PROGRAM P_EnOcean
VAR
	fbKL6581			: FB_KL6581;
	stKL6581_in  AT %I* : KL6581_INPUT;
	stKL6581_out AT %Q*	: KL6581_OUTPUT;
	stKL6581			: STR_KL6581;
	bInitCom			: BOOL := TRUE;
	
	arrEnOcean_Search	: ARRAY [1..8] OF FB_EnOcean_Search;
	nSearchIdx			: BYTE;
	bSerach				: BOOL;
	arrDevices			: ARRAY [1..8] OF INT;
	arrID				: ARRAY [1..8, 0..255] OF DWORD;
	
		//Trykknapper Atrium
	fbAtriumNiveau_Tryk_PladeB				: FB_Rec_RPS_Switch;
	fbAtriumNiveau_Tryk_Sevice				: FB_Rec_RPS_Switch;			

	//Trykknapper på gange

	
	//Trykknapper i rum
fbRum_1_111_Tryk						: FB_Rec_RPS_Switch;

END_VAR

VAR CONSTANT
	byNode_1: BYTE := 1;
	byNode_2: BYTE := 2;
	byNode_3: BYTE := 3;
	byNode_4: BYTE := 4;
	byNode_5: BYTE := 5;
	byNode_6: BYTE := 6;
	byNode_7: BYTE := 7;
	byNode_8: BYTE := 8;
END_VAR


(* Kommunikation mit der KL6581. *)
(* Communication with the KL6581. *)
fbKL6581(
	bInit			:= bInitCom,
	nIdx			:= 2,
	stKL6581_in		:= stKL6581_In,
	stKL6581_out	:= stKL6581_Out,
	bReady			=> ,
	bBusy			=> ,
	bError			=> ,
	iErrorID		=> ,
	str_KL6581		=> stKL6581);

GVL_AHDataModbus.EnOceanError	:= TO_UINT(fbKL6581.iErrorID);
(* Warten bis der Kommunikationsbaustein initialisiert wurde.*)
(* Wait until the communication function block has been initialized. *)
IF (NOT fbKL6581.bReady) THEN
	RETURN;
END_IF

FOR nSearchIdx:= 1 TO 8 DO
	arrEnOcean_Search[nSearchIdx](
		bStart:= TRUE, 
		str_KL6581:= stKL6581 , 
		byNode:= nSearchIdx, 
		bReceive=> , 
		iDevices=>arrDevices[nSearchIdx] , 
		ar_ID=> );
		
		MEMCPY(ADR(arrID[nSearchIdx,0]), ADR(arrEnOcean_Search[nSearchIdx].ar_ID), SIZEOF(arrEnOcean_Search[nSearchIdx].ar_ID)); 
END_FOR

//Gange



//RUM
 //
P_Rum_1_111();

//AtriumNiveau
A_AtriumNiveau();

ACTION A_AtriumNiveau:
fbAtriumNiveau_Tryk_PladeB(
	str_KL6581:=stKL6581 , 
	byNode:=0, 
	dw_ID:= 16#0029B92D, 
	str_EnOceanSwitch=> GVL_EnOcean.strEnOceanSwitch_AtriumNiveau_PladeB,
	by_Node=> , 
	bReceive=> );

//knap 2 
(*
fbAtriumNiveau_Tryk_Sevice(
	str_KL6581:=stKL6581 , 
	byNode:=0, 
	dw_ID:= 16#00FEE4FE87, 
	str_EnOceanSwitch=> GVL_EnOcean.strEnOceanSwitch_AtriumNiveau_Service, 
	by_Node=> , 
	bReceive=> );
*)


//Den rigtigt: 16#0029B92D
END_ACTION

ACTION P_Rum_1_111:
fbRum_1_111_Tryk(
	str_KL6581:=stKL6581 , 
	byNode:=0 , 
	dw_ID:=  16#0029ABB1, 
	str_EnOceanSwitch=> GVL_EnOcean.strEnOceanSwitch_Rum_1_111, 
	by_Node=> , 
	bReceive=> );
	
fbRum_1_111_Tryk(
	str_KL6581:=stKL6581 , 
	byNode:=0 , 
	dw_ID:=  16#0029AB7A, 
	str_EnOceanSwitch=> GVL_EnOcean.strEnOceanSwitch_Rum_1_111, 
	by_Node=> , 
	bReceive=> );
END_ACTION

ACTION P_Rum_5_454:
(*fbRum_5_454_Tryk(
	str_KL6581:=stKL6581 , 
	byNode:=4 , 
	dw_ID:=  16#0029B75D, 
	str_EnOceanSwitch=> GVL_EnOcean.strEnOceanSwitch_Rum_5_454, 
	by_Node=> , 
	bReceive=> );
*)
END_ACTION

END_PROGRAM

(* stored: Version 1.1.0.1
   POU P_EnOcean: Id {d2583012-7b8d-42b3-930e-7213eee0e992}, SpecialFunc None
   Action A_AtriumNiveau: Id {5b863a8e-6cff-4511-86bf-f0a83cf94e37}
   Action P_Rum_1_111: Id {f1d32277-aefa-4240-b07d-298bdb9f0cce}
   Action P_Rum_5_454: Id {2538d29c-9c58-4aab-9b41-90c5560a5c5d} *)
